# EPICS autosave request: iocBoot/ioc13bma/auto_positions.req
file "CARS_24_motor_positions.req", P=$(P)
file "CARS_motor_positions.req",    P=$(P), M=m25
